// TIA Portal V20 export
// export: Created 2025-12-01T14:56:59.5537053Z, ExportSetting None, DisplayName Totally Integrated Automation Portal, DisplayVersion V20 Update 3, DisplayName TIA Portal Openness, DisplayVersion V20 Update 3, DisplayName TIA Portal Version Control Interface, DisplayVersion V20 Update 3, DisplayName STEP 7 Professional, DisplayVersion V20 Update 3, DisplayName STEP 7 Safety, DisplayVersion V20 Update 2, DisplayName WinCC Basic/Comfort/Advanced, DisplayVersion V20 Update 3, DisplayName WinCC Professional, DisplayVersion V20 Update 3, DisplayName WinCC Unified, DisplayVersion V20 Update 3
FUNCTION "FC421_TL_ZPA_Tarjeta_CB_E1E3S1S3" : Void   // FC421, LAD
{ S7_Optimized_Access := 'FALSE' }
AUTHOR : TLigero
NAME : 20160208
VERSION : 3.1
// FECHA:    27/07/2014  AUTOR: G.Martin
// INSTALACION: Magyar Posta
// //////////////////////////////////
// // Registro Incidencias   ////////
// //////////////////////////////////
// FECHA:21/10/14   AUTOR MODIFICACION: N.Rodriguez
// DESCRIPCION: 
// Adaptación de la función al estandar actual
// 
// FECHA:   AUTOR MODIFICACION: 
// DESCRIPCION:
// stored: AutoNumber false, SetENOAutomatically false
   VAR_INPUT
      Mesa : UInt;
      En_Tension : Bool;
      Phs_Tx_E1 : Bool;
      Phs_Tx_E3 : Bool;
      Avance_E1 : Bool;
      Avance_E3 : Bool;
      Termico_Tx : Bool;   // Señal de termico OK
      Simul_Mx : Bool;
      Invertir_Sentido : Bool;   // OFF sentido 1-3 a ON sentido 3-1
      AVTF_Ent_M1 : Bool;
      AVTF_Ent_M3 : Bool;
      PTF_Sal_M3 : Bool;
      NXT_Avance_M3 : Bool;
      PTF_Sal_M1 : Bool;
      NXT_Avance_M1 : Bool;
      V_CNT_pHsMx_E1 : UDInt;
      V_CNT_pHsMx_E3 : UDInt;
      V_Gap_E1 : UDInt;
      V_Gap_E3 : UDInt;
      V_Paro : UDInt;
      V_TOut_Tx_Mx : UDInt;
      V_Salida : UDInt;
   END_VAR
   VAR_OUTPUT
      PTF_Ent_M1 : Bool;
      PTF_Ent_M3 : Bool;
      AVTF_Sal_M1 : Bool;
      NXT_Descarga_Act_M1 : Bool;
      AVTF_Sal_M3 : Bool;
      NXT_Descarga_Act_M3 : Bool;
   END_VAR
   VAR_IN_OUT
      Mem_CNT_Salida : Bool;
      Mem_CNT_Tmp_Paro_Tx : Bool;
      MAUX_FP_Marcha : Bool;
      MAUX_FN_PHS : Bool;
      MAUX_FP_Direc : Bool;
      MAUX_FN_Direc : Bool;
   END_VAR
   VAR_TEMP
      OK_Avance : Bool;
      fp_Marcha : Bool;
      fn_phs_tx : Bool;
      fp_phs_tx : Bool;
      Mem_CNT_Centrado : Bool;
      Mem_CNT_Gap : Bool;
      fp_direc : Bool;
      fn_direc : Bool;
      Error_Atasco : Bool;
      Error_Atasco_Inv : Bool;
      TEMP_NXT_AVTF : Bool;
      TEMP_NXT_AVTF_Inv : Bool;
      ok_tension : Bool;
   END_VAR
   VAR_TEMP   // added for the SCL form of the ladder/FBD networks
      _w1 : Bool;
      _w2 : Bool;
   END_VAR
BEGIN

REGION Network 1: Marca General Error
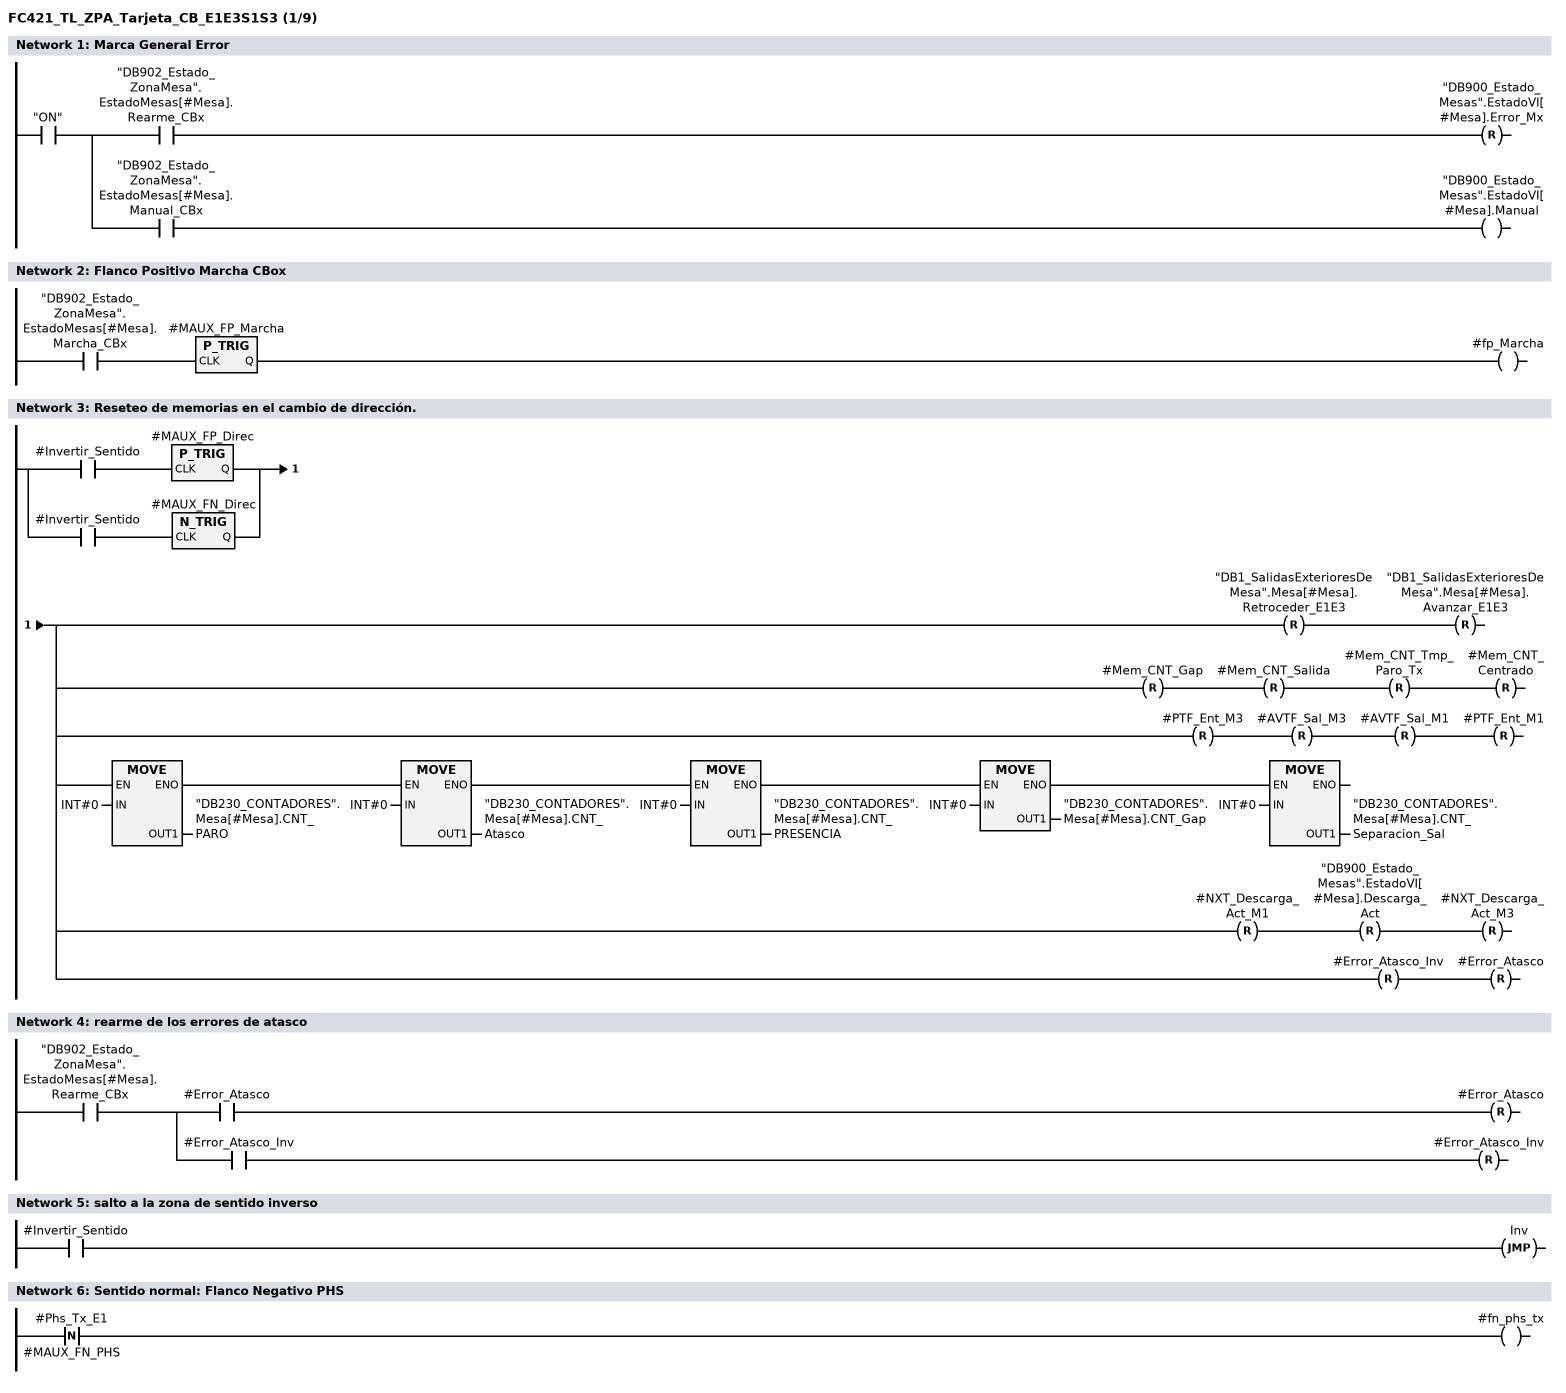
   RUNG wire#powerrail
      Contact( "ON" )
      wire#w1
      Contact( "DB902_Estado_ZonaMesa".EstadoMesas[#Mesa].Rearme_CBx )
      R_Coil( "DB900_Estado_Mesas".EstadoVI[#Mesa].Error_Mx )
   END_RUNG
   RUNG wire#w1
      Contact( "DB902_Estado_ZonaMesa".EstadoMesas[#Mesa].Manual_CBx )
      Coil( "DB900_Estado_Mesas".EstadoVI[#Mesa].Manual )
   END_RUNG
   // the same network as SCL:
   IF "ON" AND "DB902_Estado_ZonaMesa".EstadoMesas[#Mesa].Rearme_CBx THEN
       "DB900_Estado_Mesas".EstadoVI[#Mesa].Error_Mx := FALSE;
   END_IF;
   "DB900_Estado_Mesas".EstadoVI[#Mesa].Manual := "ON" AND "DB902_Estado_ZonaMesa".EstadoMesas[#Mesa].Manual_CBx;
END_REGION

REGION Network 2: Flanco Positivo Marcha CBox
   RUNG wire#powerrail
      Contact( "DB902_Estado_ZonaMesa".EstadoMesas[#Mesa].Marcha_CBx )
      P_Trig( #MAUX_FP_Marcha )
      Coil( #fp_Marcha )
   END_RUNG
   // the same network as SCL:
   #_w1 := "DB902_Estado_ZonaMesa".EstadoMesas[#Mesa].Marcha_CBx AND NOT #MAUX_FP_Marcha;   // rising edge
   #MAUX_FP_Marcha := "DB902_Estado_ZonaMesa".EstadoMesas[#Mesa].Marcha_CBx;
   #fp_Marcha := #_w1;
END_REGION

REGION Network 3: Reseteo de memorias en el cambio de dirección.
   RUNG wire#powerrail
      Contact( #Invertir_Sentido )
      P_Trig( #MAUX_FP_Direc )
      wire#w1
      R_Coil( "DB1_SalidasExterioresDeMesa".Mesa[#Mesa].Retroceder_E1E3 )
      R_Coil( "DB1_SalidasExterioresDeMesa".Mesa[#Mesa].Avanzar_E1E3 )
   END_RUNG
   RUNG wire#powerrail
      Contact( #Invertir_Sentido )
      N_Trig( #MAUX_FN_Direc )
   END_RUNG wire#w1
   RUNG wire#w1
      R_Coil( #Mem_CNT_Gap )
      R_Coil( #Mem_CNT_Salida )
      R_Coil( #Mem_CNT_Tmp_Paro_Tx )
      R_Coil( #Mem_CNT_Centrado )
   END_RUNG
   RUNG wire#w1
      R_Coil( #PTF_Ent_M3 )
      R_Coil( #AVTF_Sal_M3 )
      R_Coil( #AVTF_Sal_M1 )
      R_Coil( #PTF_Ent_M1 )
   END_RUNG
   RUNG wire#w1
      { S7_GenerateENO := "TRUE" } Move(in := INT#0, out1 => "DB230_CONTADORES".Mesa[#Mesa].CNT_PARO)
      { S7_GenerateENO := "TRUE" } Move(in := INT#0, out1 => "DB230_CONTADORES".Mesa[#Mesa].CNT_Atasco)
      { S7_GenerateENO := "TRUE" } Move(in := INT#0, out1 => "DB230_CONTADORES".Mesa[#Mesa].CNT_PRESENCIA)
      { S7_GenerateENO := "TRUE" } Move(in := INT#0, out1 => "DB230_CONTADORES".Mesa[#Mesa].CNT_Gap)
      { S7_GenerateENO := "TRUE" } Move(in := INT#0, out1 => "DB230_CONTADORES".Mesa[#Mesa].CNT_Separacion_Sal)
   END_RUNG
   RUNG wire#w1
      R_Coil( #NXT_Descarga_Act_M1 )
      R_Coil( "DB900_Estado_Mesas".EstadoVI[#Mesa].Descarga_Act )
      R_Coil( #NXT_Descarga_Act_M3 )
   END_RUNG
   RUNG wire#w1
      R_Coil( #Error_Atasco_Inv )
      R_Coil( #Error_Atasco )
   END_RUNG
   // the same network as SCL:
   // ENO of a box is taken as its EN; it also drops when the box reports an error
   #_w1 := #Invertir_Sentido AND NOT #MAUX_FP_Direc;   // rising edge
   #MAUX_FP_Direc := #Invertir_Sentido;
   #_w2 := NOT #Invertir_Sentido AND #MAUX_FN_Direc;   // falling edge
   #MAUX_FN_Direc := #Invertir_Sentido;
   IF #_w1 OR #_w2 THEN
       "DB1_SalidasExterioresDeMesa".Mesa[#Mesa].Retroceder_E1E3 := FALSE;
       "DB1_SalidasExterioresDeMesa".Mesa[#Mesa].Avanzar_E1E3 := FALSE;
       #Mem_CNT_Gap := FALSE;
       #Mem_CNT_Salida := FALSE;
       #Mem_CNT_Tmp_Paro_Tx := FALSE;
       #Mem_CNT_Centrado := FALSE;
       #PTF_Ent_M3 := FALSE;
       #AVTF_Sal_M3 := FALSE;
       #AVTF_Sal_M1 := FALSE;
       #PTF_Ent_M1 := FALSE;
       "DB230_CONTADORES".Mesa[#Mesa].CNT_PARO := INT#0;
       "DB230_CONTADORES".Mesa[#Mesa].CNT_Atasco := INT#0;
       "DB230_CONTADORES".Mesa[#Mesa].CNT_PRESENCIA := INT#0;
       "DB230_CONTADORES".Mesa[#Mesa].CNT_Gap := INT#0;
       "DB230_CONTADORES".Mesa[#Mesa].CNT_Separacion_Sal := INT#0;
       #NXT_Descarga_Act_M1 := FALSE;
       "DB900_Estado_Mesas".EstadoVI[#Mesa].Descarga_Act := FALSE;
       #NXT_Descarga_Act_M3 := FALSE;
       #Error_Atasco_Inv := FALSE;
       #Error_Atasco := FALSE;
   END_IF;
END_REGION

REGION Network 4: rearme de los errores de atasco
   RUNG wire#powerrail
      Contact( "DB902_Estado_ZonaMesa".EstadoMesas[#Mesa].Rearme_CBx )
      wire#w1
      Contact( #Error_Atasco )
      R_Coil( #Error_Atasco )
   END_RUNG
   RUNG wire#w1
      Contact( #Error_Atasco_Inv )
      R_Coil( #Error_Atasco_Inv )
   END_RUNG
   // the same network as SCL:
   IF "DB902_Estado_ZonaMesa".EstadoMesas[#Mesa].Rearme_CBx AND #Error_Atasco THEN
       #Error_Atasco := FALSE;
   END_IF;
   IF "DB902_Estado_ZonaMesa".EstadoMesas[#Mesa].Rearme_CBx AND #Error_Atasco_Inv THEN
       #Error_Atasco_Inv := FALSE;
   END_IF;
END_REGION

REGION Network 5: salto a la zona de sentido inverso
   RUNG wire#powerrail
      Contact( #Invertir_Sentido )
      JumpCoil( Inv )
   END_RUNG
   // the same network as SCL:
   IF #Invertir_Sentido THEN GOTO Inv; END_IF;
END_REGION

REGION Network 6: Sentido normal: Flanco Negativo PHS
   RUNG wire#powerrail
      N_Contact(operand := #Phs_Tx_E1, bit := #MAUX_FN_PHS)
      Coil( #fn_phs_tx )
   END_RUNG
   // the same network as SCL:
   #_w1 := NOT #Phs_Tx_E1 AND #MAUX_FN_PHS;   // falling edge of #Phs_Tx_E1
   #MAUX_FN_PHS := #Phs_Tx_E1;
   #fn_phs_tx := #_w1;
END_REGION

REGION Network 7: En Tension
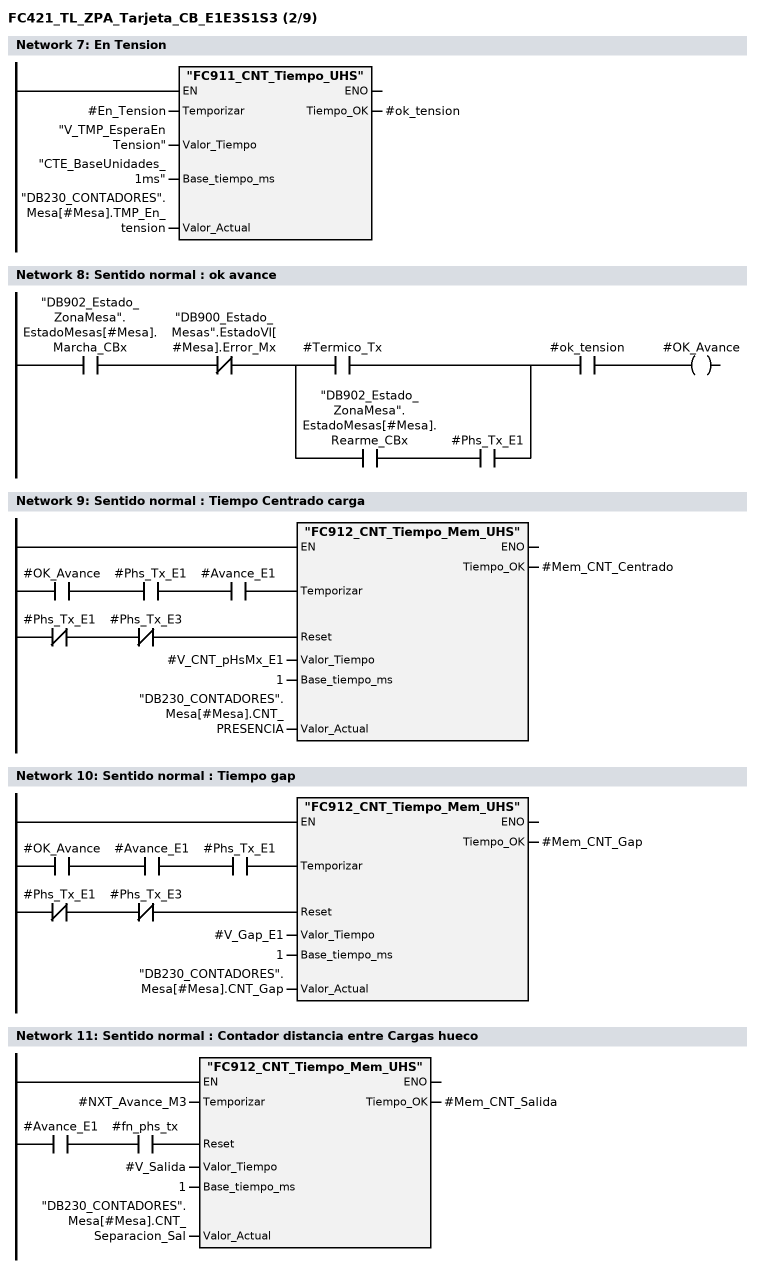
   RUNG wire#powerrail
      "FC911_CNT_Tiempo_UHS"(Temporizar := #En_Tension, Valor_Tiempo := "V_TMP_EsperaEnTension", Base_tiempo_ms := "CTE_BaseUnidades_1ms", Valor_Actual := "DB230_CONTADORES".Mesa[#Mesa].TMP_En_tension, Tiempo_OK => #ok_tension)
   END_RUNG
   // the same network as SCL:
   "FC911_CNT_Tiempo_UHS"(Temporizar := #En_Tension,
                          Valor_Tiempo := "V_TMP_EsperaEnTension",
                          Base_tiempo_ms := "CTE_BaseUnidades_1ms",
                          Valor_Actual := "DB230_CONTADORES".Mesa[#Mesa].TMP_En_tension,
                          Tiempo_OK => #ok_tension);
END_REGION

REGION Network 8: Sentido normal : ok avance
   RUNG wire#powerrail
      Contact( "DB902_Estado_ZonaMesa".EstadoMesas[#Mesa].Marcha_CBx )
      I_Contact( "DB900_Estado_Mesas".EstadoVI[#Mesa].Error_Mx )
      wire#w1
      Contact( #Termico_Tx )
      wire#w2
      Contact( #ok_tension )
      Coil( #OK_Avance )
   END_RUNG
   RUNG wire#w1
      Contact( "DB902_Estado_ZonaMesa".EstadoMesas[#Mesa].Rearme_CBx )
      Contact( #Phs_Tx_E1 )
   END_RUNG wire#w2
   // the same network as SCL:
   #OK_Avance := "DB902_Estado_ZonaMesa".EstadoMesas[#Mesa].Marcha_CBx AND NOT "DB900_Estado_Mesas".EstadoVI[#Mesa].Error_Mx AND (#Termico_Tx OR ("DB902_Estado_ZonaMesa".EstadoMesas[#Mesa].Rearme_CBx AND #Phs_Tx_E1)) AND #ok_tension;
END_REGION

REGION Network 9: Sentido normal : Tiempo Centrado carga
   RUNG wire#powerrail
      "FC912_CNT_Tiempo_Mem_UHS"(Temporizar := wire#w1, Reset := wire#w2, Valor_Tiempo := #V_CNT_pHsMx_E1, Base_tiempo_ms := 1, Valor_Actual := "DB230_CONTADORES".Mesa[#Mesa].CNT_PRESENCIA, Tiempo_OK => #Mem_CNT_Centrado)
   END_RUNG
   RUNG wire#powerrail
      Contact( #OK_Avance )
      Contact( #Phs_Tx_E1 )
      Contact( #Avance_E1 )
   END_RUNG wire#w1
   RUNG wire#powerrail
      I_Contact( #Phs_Tx_E1 )
      I_Contact( #Phs_Tx_E3 )
   END_RUNG wire#w2
   // the same network as SCL:
   "FC912_CNT_Tiempo_Mem_UHS"(Temporizar := #OK_Avance AND #Phs_Tx_E1 AND #Avance_E1,
                           Reset := NOT #Phs_Tx_E1 AND NOT #Phs_Tx_E3,
                           Valor_Tiempo := #V_CNT_pHsMx_E1,
                           Base_tiempo_ms := 1,
                           Valor_Actual := "DB230_CONTADORES".Mesa[#Mesa].CNT_PRESENCIA,
                           Tiempo_OK => #Mem_CNT_Centrado);
END_REGION

REGION Network 10: Sentido normal : Tiempo gap
   RUNG wire#powerrail
      "FC912_CNT_Tiempo_Mem_UHS"(Temporizar := wire#w1, Reset := wire#w2, Valor_Tiempo := #V_Gap_E1, Base_tiempo_ms := 1, Valor_Actual := "DB230_CONTADORES".Mesa[#Mesa].CNT_Gap, Tiempo_OK => #Mem_CNT_Gap)
   END_RUNG
   RUNG wire#powerrail
      Contact( #OK_Avance )
      Contact( #Avance_E1 )
      Contact( #Phs_Tx_E1 )
   END_RUNG wire#w1
   RUNG wire#powerrail
      I_Contact( #Phs_Tx_E1 )
      I_Contact( #Phs_Tx_E3 )
   END_RUNG wire#w2
   // the same network as SCL:
   "FC912_CNT_Tiempo_Mem_UHS"(Temporizar := #OK_Avance AND #Avance_E1 AND #Phs_Tx_E1,
                           Reset := NOT #Phs_Tx_E1 AND NOT #Phs_Tx_E3,
                           Valor_Tiempo := #V_Gap_E1,
                           Base_tiempo_ms := 1,
                           Valor_Actual := "DB230_CONTADORES".Mesa[#Mesa].CNT_Gap,
                           Tiempo_OK => #Mem_CNT_Gap);
END_REGION

REGION Network 11: Sentido normal : Contador distancia entre Cargas hueco
   RUNG wire#powerrail
      "FC912_CNT_Tiempo_Mem_UHS"(Reset := wire#w1, Temporizar := #NXT_Avance_M3, Valor_Tiempo := #V_Salida, Base_tiempo_ms := 1, Valor_Actual := "DB230_CONTADORES".Mesa[#Mesa].CNT_Separacion_Sal, Tiempo_OK => #Mem_CNT_Salida)
   END_RUNG
   RUNG wire#powerrail
      Contact( #Avance_E1 )
      Contact( #fn_phs_tx )
   END_RUNG wire#w1
   // the same network as SCL:
   "FC912_CNT_Tiempo_Mem_UHS"(Temporizar := #NXT_Avance_M3,
                           Reset := #Avance_E1 AND #fn_phs_tx,
                           Valor_Tiempo := #V_Salida,
                           Base_tiempo_ms := 1,
                           Valor_Actual := "DB230_CONTADORES".Mesa[#Mesa].CNT_Separacion_Sal,
                           Tiempo_OK => #Mem_CNT_Salida);
END_REGION

REGION Network 12: Sentido normal : temporizador de paro
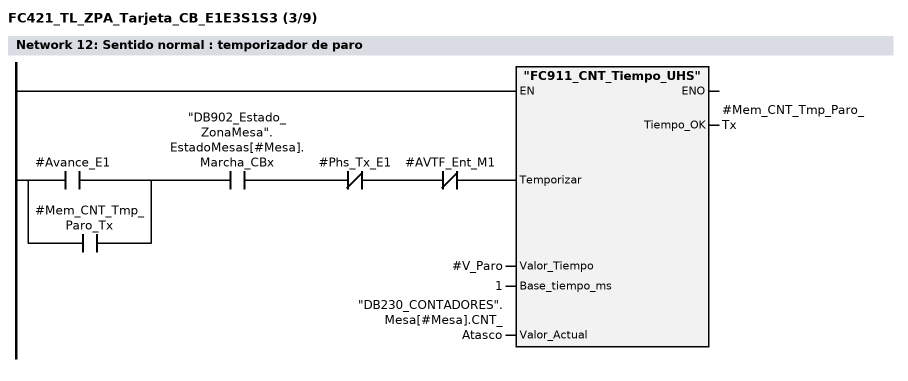
   RUNG wire#powerrail
      "FC911_CNT_Tiempo_UHS"(Temporizar := wire#w2, Valor_Tiempo := #V_Paro, Base_tiempo_ms := 1, Valor_Actual := "DB230_CONTADORES".Mesa[#Mesa].CNT_Atasco, Tiempo_OK => #Mem_CNT_Tmp_Paro_Tx)
   END_RUNG
   RUNG wire#powerrail
      Contact( #Avance_E1 )
      wire#w1
      Contact( "DB902_Estado_ZonaMesa".EstadoMesas[#Mesa].Marcha_CBx )
      I_Contact( #Phs_Tx_E1 )
      I_Contact( #AVTF_Ent_M1 )
   END_RUNG wire#w2
   RUNG wire#powerrail
      Contact( #Mem_CNT_Tmp_Paro_Tx )
   END_RUNG wire#w1
   // the same network as SCL:
   "FC911_CNT_Tiempo_UHS"(Temporizar := (#Avance_E1 OR #Mem_CNT_Tmp_Paro_Tx) AND "DB902_Estado_ZonaMesa".EstadoMesas[#Mesa].Marcha_CBx AND NOT #Phs_Tx_E1 AND NOT #AVTF_Ent_M1,
                          Valor_Tiempo := #V_Paro,
                          Base_tiempo_ms := 1,
                          Valor_Actual := "DB230_CONTADORES".Mesa[#Mesa].CNT_Atasco,
                          Tiempo_OK => #Mem_CNT_Tmp_Paro_Tx);
END_REGION

REGION Network 13: Sentido normal : avance 13
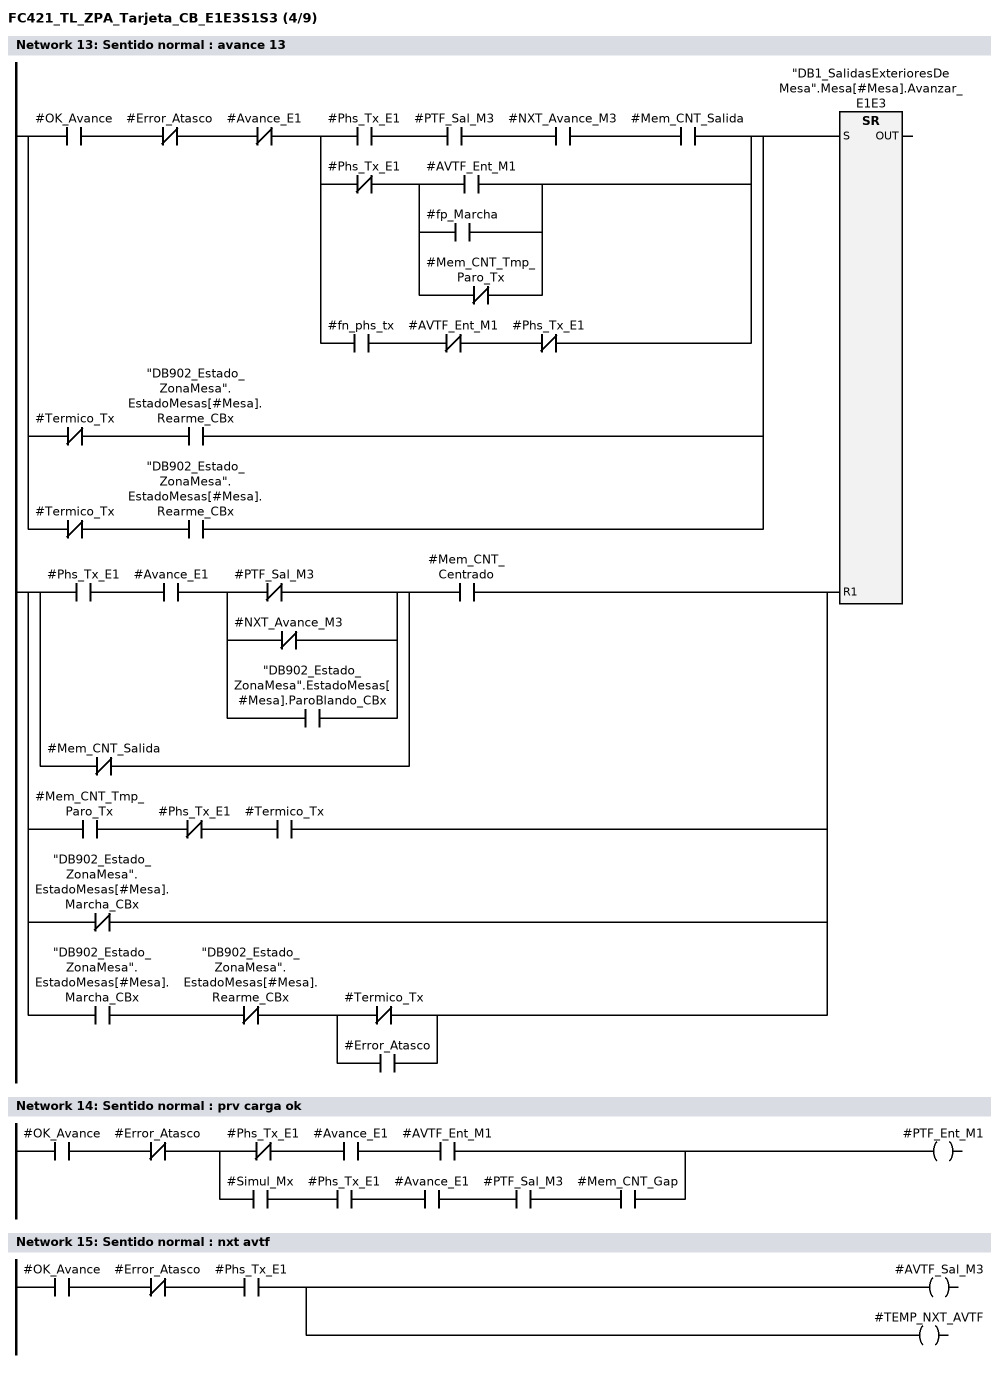
   RUNG wire#powerrail
      Contact( #OK_Avance )
      I_Contact( #Error_Atasco )
      I_Contact( #Avance_E1 )
      wire#w1
      Contact( #Phs_Tx_E1 )
      Contact( #PTF_Sal_M3 )
      Contact( #NXT_Avance_M3 )
      Contact( #Mem_CNT_Salida )
      wire#w2
      S_SR(operand := "DB1_SalidasExterioresDeMesa".Mesa[#Mesa].Avanzar_E1E3, r1 := wire#w7)
   END_RUNG
   RUNG wire#w1
      I_Contact( #Phs_Tx_E1 )
      wire#w3
      Contact( #AVTF_Ent_M1 )
   END_RUNG wire#w2
   RUNG wire#w3
      Contact( #fp_Marcha )
   END_RUNG wire#w2
   RUNG wire#w3
      I_Contact( #Mem_CNT_Tmp_Paro_Tx )
   END_RUNG wire#w2
   RUNG wire#w1
      Contact( #fn_phs_tx )
      I_Contact( #AVTF_Ent_M1 )
      I_Contact( #Phs_Tx_E1 )
   END_RUNG wire#w2
   RUNG wire#powerrail
      I_Contact( #Termico_Tx )
      Contact( "DB902_Estado_ZonaMesa".EstadoMesas[#Mesa].Rearme_CBx )
   END_RUNG wire#w2
   RUNG wire#powerrail
      I_Contact( #Termico_Tx )
      Contact( "DB902_Estado_ZonaMesa".EstadoMesas[#Mesa].Rearme_CBx )
   END_RUNG wire#w2
   RUNG wire#powerrail
      Contact( #Phs_Tx_E1 )
      Contact( #Avance_E1 )
      wire#w4
      I_Contact( #PTF_Sal_M3 )
      wire#w5
      Contact( #Mem_CNT_Centrado )
   END_RUNG wire#w7
   RUNG wire#w4
      I_Contact( #NXT_Avance_M3 )
   END_RUNG wire#w5
   RUNG wire#w4
      Contact( "DB902_Estado_ZonaMesa".EstadoMesas[#Mesa].ParoBlando_CBx )
   END_RUNG wire#w5
   RUNG wire#powerrail
      I_Contact( #Mem_CNT_Salida )
   END_RUNG wire#w5
   RUNG wire#powerrail
      Contact( #Mem_CNT_Tmp_Paro_Tx )
      I_Contact( #Phs_Tx_E1 )
      Contact( #Termico_Tx )
   END_RUNG wire#w7
   RUNG wire#powerrail
      I_Contact( "DB902_Estado_ZonaMesa".EstadoMesas[#Mesa].Marcha_CBx )
   END_RUNG wire#w7
   RUNG wire#powerrail
      Contact( "DB902_Estado_ZonaMesa".EstadoMesas[#Mesa].Marcha_CBx )
      I_Contact( "DB902_Estado_ZonaMesa".EstadoMesas[#Mesa].Rearme_CBx )
      wire#w6
      I_Contact( #Termico_Tx )
   END_RUNG wire#w7
   RUNG wire#w6
      Contact( #Error_Atasco )
   END_RUNG wire#w7
   // the same network as SCL:
   #_w1 := (((#Phs_Tx_E1 AND #Avance_E1 AND (NOT #PTF_Sal_M3 OR NOT #NXT_Avance_M3 OR "DB902_Estado_ZonaMesa".EstadoMesas[#Mesa].ParoBlando_CBx)) OR NOT #Mem_CNT_Salida) AND #Mem_CNT_Centrado) OR (#Mem_CNT_Tmp_Paro_Tx AND NOT #Phs_Tx_E1 AND #Termico_Tx) OR NOT "DB902_Estado_ZonaMesa".EstadoMesas[#Mesa].Marcha_CBx OR ("DB902_Estado_ZonaMesa".EstadoMesas[#Mesa].Marcha_CBx AND NOT "DB902_Estado_ZonaMesa".EstadoMesas[#Mesa].Rearme_CBx AND (NOT #Termico_Tx OR #Error_Atasco));
   IF (#OK_Avance AND NOT #Error_Atasco AND NOT #Avance_E1 AND ((#Phs_Tx_E1 AND #PTF_Sal_M3 AND #NXT_Avance_M3 AND #Mem_CNT_Salida) OR (NOT #Phs_Tx_E1 AND (#AVTF_Ent_M1 OR #fp_Marcha OR NOT #Mem_CNT_Tmp_Paro_Tx)) OR (#fn_phs_tx AND NOT #AVTF_Ent_M1 AND NOT #Phs_Tx_E1))) OR (NOT #Termico_Tx AND "DB902_Estado_ZonaMesa".EstadoMesas[#Mesa].Rearme_CBx) OR (NOT #Termico_Tx AND "DB902_Estado_ZonaMesa".EstadoMesas[#Mesa].Rearme_CBx) THEN
       "DB1_SalidasExterioresDeMesa".Mesa[#Mesa].Avanzar_E1E3 := TRUE;   // SR flip-flop
   END_IF;
   IF #_w1 THEN "DB1_SalidasExterioresDeMesa".Mesa[#Mesa].Avanzar_E1E3 := FALSE; END_IF;
END_REGION

REGION Network 14: Sentido normal : prv carga ok
   RUNG wire#powerrail
      Contact( #OK_Avance )
      I_Contact( #Error_Atasco )
      wire#w1
      I_Contact( #Phs_Tx_E1 )
      Contact( #Avance_E1 )
      Contact( #AVTF_Ent_M1 )
      wire#w2
      Coil( #PTF_Ent_M1 )
   END_RUNG
   RUNG wire#w1
      Contact( #Simul_Mx )
      Contact( #Phs_Tx_E1 )
      Contact( #Avance_E1 )
      Contact( #PTF_Sal_M3 )
      Contact( #Mem_CNT_Gap )
   END_RUNG wire#w2
   // the same network as SCL:
   #PTF_Ent_M1 := #OK_Avance AND NOT #Error_Atasco AND ((NOT #Phs_Tx_E1 AND #Avance_E1 AND #AVTF_Ent_M1) OR (#Simul_Mx AND #Phs_Tx_E1 AND #Avance_E1 AND #PTF_Sal_M3 AND #Mem_CNT_Gap));
END_REGION

REGION Network 15: Sentido normal : nxt avtf
   RUNG wire#powerrail
      Contact( #OK_Avance )
      I_Contact( #Error_Atasco )
      Contact( #Phs_Tx_E1 )
      wire#w1
      Coil( #AVTF_Sal_M3 )
   END_RUNG
   RUNG wire#w1
      Coil( #TEMP_NXT_AVTF )
   END_RUNG
   // the same network as SCL:
   #AVTF_Sal_M3 := #OK_Avance AND NOT #Error_Atasco AND #Phs_Tx_E1;
   #TEMP_NXT_AVTF := #AVTF_Sal_M3;
END_REGION

REGION Network 16: Sentido normal : nxt descarga activa
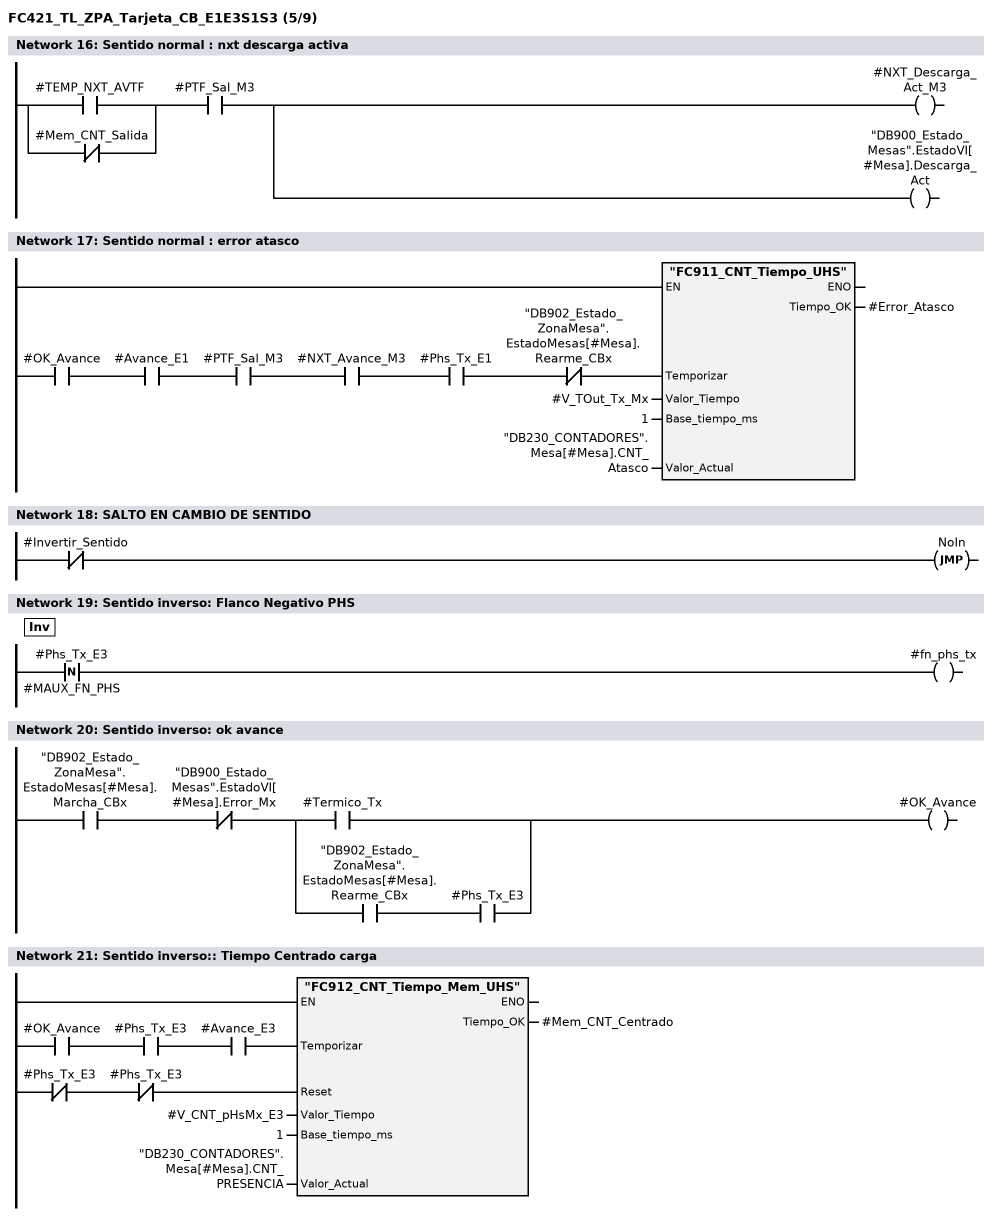
   RUNG wire#powerrail
      Contact( #TEMP_NXT_AVTF )
      wire#w1
      Contact( #PTF_Sal_M3 )
      wire#w2
      Coil( #NXT_Descarga_Act_M3 )
   END_RUNG
   RUNG wire#powerrail
      I_Contact( #Mem_CNT_Salida )
   END_RUNG wire#w1
   RUNG wire#w2
      Coil( "DB900_Estado_Mesas".EstadoVI[#Mesa].Descarga_Act )
   END_RUNG
   // the same network as SCL:
   #NXT_Descarga_Act_M3 := (#TEMP_NXT_AVTF OR NOT #Mem_CNT_Salida) AND #PTF_Sal_M3;
   "DB900_Estado_Mesas".EstadoVI[#Mesa].Descarga_Act := #NXT_Descarga_Act_M3;
END_REGION

REGION Network 17: Sentido normal : error atasco
   RUNG wire#powerrail
      "FC911_CNT_Tiempo_UHS"(Temporizar := wire#w1, Valor_Tiempo := #V_TOut_Tx_Mx, Base_tiempo_ms := 1, Valor_Actual := "DB230_CONTADORES".Mesa[#Mesa].CNT_Atasco, Tiempo_OK => #Error_Atasco)
   END_RUNG
   RUNG wire#powerrail
      Contact( #OK_Avance )
      Contact( #Avance_E1 )
      Contact( #PTF_Sal_M3 )
      Contact( #NXT_Avance_M3 )
      Contact( #Phs_Tx_E1 )
      I_Contact( "DB902_Estado_ZonaMesa".EstadoMesas[#Mesa].Rearme_CBx )
   END_RUNG wire#w1
   // the same network as SCL:
   "FC911_CNT_Tiempo_UHS"(Temporizar := #OK_Avance AND #Avance_E1 AND #PTF_Sal_M3 AND #NXT_Avance_M3 AND #Phs_Tx_E1 AND NOT "DB902_Estado_ZonaMesa".EstadoMesas[#Mesa].Rearme_CBx,
                          Valor_Tiempo := #V_TOut_Tx_Mx,
                          Base_tiempo_ms := 1,
                          Valor_Actual := "DB230_CONTADORES".Mesa[#Mesa].CNT_Atasco,
                          Tiempo_OK => #Error_Atasco);
END_REGION

REGION Network 18: SALTO EN CAMBIO DE SENTIDO
   RUNG wire#powerrail
      I_Contact( #Invertir_Sentido )
      JumpCoil( NoIn )
   END_RUNG
   // the same network as SCL:
   IF NOT #Invertir_Sentido THEN GOTO NoIn; END_IF;
END_REGION

REGION Network 19: Sentido inverso: Flanco Negativo PHS
   Label( Inv )
   RUNG wire#powerrail
      N_Contact(operand := #Phs_Tx_E3, bit := #MAUX_FN_PHS)
      Coil( #fn_phs_tx )
   END_RUNG
   // the same network as SCL:
   Inv:
   #_w1 := NOT #Phs_Tx_E3 AND #MAUX_FN_PHS;   // falling edge of #Phs_Tx_E3
   #MAUX_FN_PHS := #Phs_Tx_E3;
   #fn_phs_tx := #_w1;
END_REGION

REGION Network 20: Sentido inverso: ok avance
   RUNG wire#powerrail
      Contact( "DB902_Estado_ZonaMesa".EstadoMesas[#Mesa].Marcha_CBx )
      I_Contact( "DB900_Estado_Mesas".EstadoVI[#Mesa].Error_Mx )
      wire#w1
      Contact( #Termico_Tx )
      wire#w2
      Coil( #OK_Avance )
   END_RUNG
   RUNG wire#w1
      Contact( "DB902_Estado_ZonaMesa".EstadoMesas[#Mesa].Rearme_CBx )
      Contact( #Phs_Tx_E3 )
   END_RUNG wire#w2
   // the same network as SCL:
   #OK_Avance := "DB902_Estado_ZonaMesa".EstadoMesas[#Mesa].Marcha_CBx AND NOT "DB900_Estado_Mesas".EstadoVI[#Mesa].Error_Mx AND (#Termico_Tx OR ("DB902_Estado_ZonaMesa".EstadoMesas[#Mesa].Rearme_CBx AND #Phs_Tx_E3));
END_REGION

REGION Network 21: Sentido inverso:: Tiempo Centrado carga
   RUNG wire#powerrail
      "FC912_CNT_Tiempo_Mem_UHS"(Temporizar := wire#w1, Reset := wire#w2, Valor_Tiempo := #V_CNT_pHsMx_E3, Base_tiempo_ms := 1, Valor_Actual := "DB230_CONTADORES".Mesa[#Mesa].CNT_PRESENCIA, Tiempo_OK => #Mem_CNT_Centrado)
   END_RUNG
   RUNG wire#powerrail
      Contact( #OK_Avance )
      Contact( #Phs_Tx_E3 )
      Contact( #Avance_E3 )
   END_RUNG wire#w1
   RUNG wire#powerrail
      I_Contact( #Phs_Tx_E3 )
      I_Contact( #Phs_Tx_E3 )
   END_RUNG wire#w2
   // the same network as SCL:
   "FC912_CNT_Tiempo_Mem_UHS"(Temporizar := #OK_Avance AND #Phs_Tx_E3 AND #Avance_E3,
                           Reset := NOT #Phs_Tx_E3 AND NOT #Phs_Tx_E3,
                           Valor_Tiempo := #V_CNT_pHsMx_E3,
                           Base_tiempo_ms := 1,
                           Valor_Actual := "DB230_CONTADORES".Mesa[#Mesa].CNT_PRESENCIA,
                           Tiempo_OK => #Mem_CNT_Centrado);
END_REGION

REGION Network 22: Sentido inverso: Tiempo gap
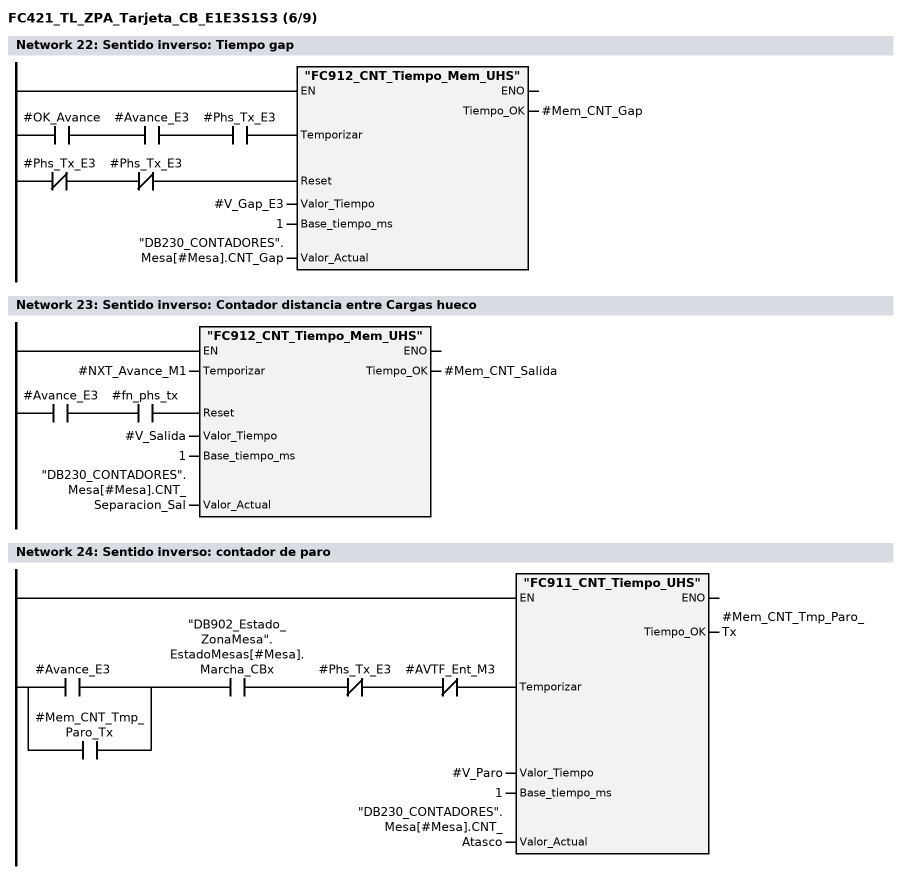
   RUNG wire#powerrail
      "FC912_CNT_Tiempo_Mem_UHS"(Temporizar := wire#w1, Reset := wire#w2, Valor_Tiempo := #V_Gap_E3, Base_tiempo_ms := 1, Valor_Actual := "DB230_CONTADORES".Mesa[#Mesa].CNT_Gap, Tiempo_OK => #Mem_CNT_Gap)
   END_RUNG
   RUNG wire#powerrail
      Contact( #OK_Avance )
      Contact( #Avance_E3 )
      Contact( #Phs_Tx_E3 )
   END_RUNG wire#w1
   RUNG wire#powerrail
      I_Contact( #Phs_Tx_E3 )
      I_Contact( #Phs_Tx_E3 )
   END_RUNG wire#w2
   // the same network as SCL:
   "FC912_CNT_Tiempo_Mem_UHS"(Temporizar := #OK_Avance AND #Avance_E3 AND #Phs_Tx_E3,
                           Reset := NOT #Phs_Tx_E3 AND NOT #Phs_Tx_E3,
                           Valor_Tiempo := #V_Gap_E3,
                           Base_tiempo_ms := 1,
                           Valor_Actual := "DB230_CONTADORES".Mesa[#Mesa].CNT_Gap,
                           Tiempo_OK => #Mem_CNT_Gap);
END_REGION

REGION Network 23: Sentido inverso: Contador distancia entre Cargas hueco
   RUNG wire#powerrail
      "FC912_CNT_Tiempo_Mem_UHS"(Reset := wire#w1, Temporizar := #NXT_Avance_M1, Valor_Tiempo := #V_Salida, Base_tiempo_ms := 1, Valor_Actual := "DB230_CONTADORES".Mesa[#Mesa].CNT_Separacion_Sal, Tiempo_OK => #Mem_CNT_Salida)
   END_RUNG
   RUNG wire#powerrail
      Contact( #Avance_E3 )
      Contact( #fn_phs_tx )
   END_RUNG wire#w1
   // the same network as SCL:
   "FC912_CNT_Tiempo_Mem_UHS"(Temporizar := #NXT_Avance_M1,
                           Reset := #Avance_E3 AND #fn_phs_tx,
                           Valor_Tiempo := #V_Salida,
                           Base_tiempo_ms := 1,
                           Valor_Actual := "DB230_CONTADORES".Mesa[#Mesa].CNT_Separacion_Sal,
                           Tiempo_OK => #Mem_CNT_Salida);
END_REGION

REGION Network 24: Sentido inverso: contador de paro
   RUNG wire#powerrail
      "FC911_CNT_Tiempo_UHS"(Temporizar := wire#w2, Valor_Tiempo := #V_Paro, Base_tiempo_ms := 1, Valor_Actual := "DB230_CONTADORES".Mesa[#Mesa].CNT_Atasco, Tiempo_OK => #Mem_CNT_Tmp_Paro_Tx)
   END_RUNG
   RUNG wire#powerrail
      Contact( #Avance_E3 )
      wire#w1
      Contact( "DB902_Estado_ZonaMesa".EstadoMesas[#Mesa].Marcha_CBx )
      I_Contact( #Phs_Tx_E3 )
      I_Contact( #AVTF_Ent_M3 )
   END_RUNG wire#w2
   RUNG wire#powerrail
      Contact( #Mem_CNT_Tmp_Paro_Tx )
   END_RUNG wire#w1
   // the same network as SCL:
   "FC911_CNT_Tiempo_UHS"(Temporizar := (#Avance_E3 OR #Mem_CNT_Tmp_Paro_Tx) AND "DB902_Estado_ZonaMesa".EstadoMesas[#Mesa].Marcha_CBx AND NOT #Phs_Tx_E3 AND NOT #AVTF_Ent_M3,
                          Valor_Tiempo := #V_Paro,
                          Base_tiempo_ms := 1,
                          Valor_Actual := "DB230_CONTADORES".Mesa[#Mesa].CNT_Atasco,
                          Tiempo_OK => #Mem_CNT_Tmp_Paro_Tx);
END_REGION

REGION Network 25: Sentido inverso: retroceso 1-3
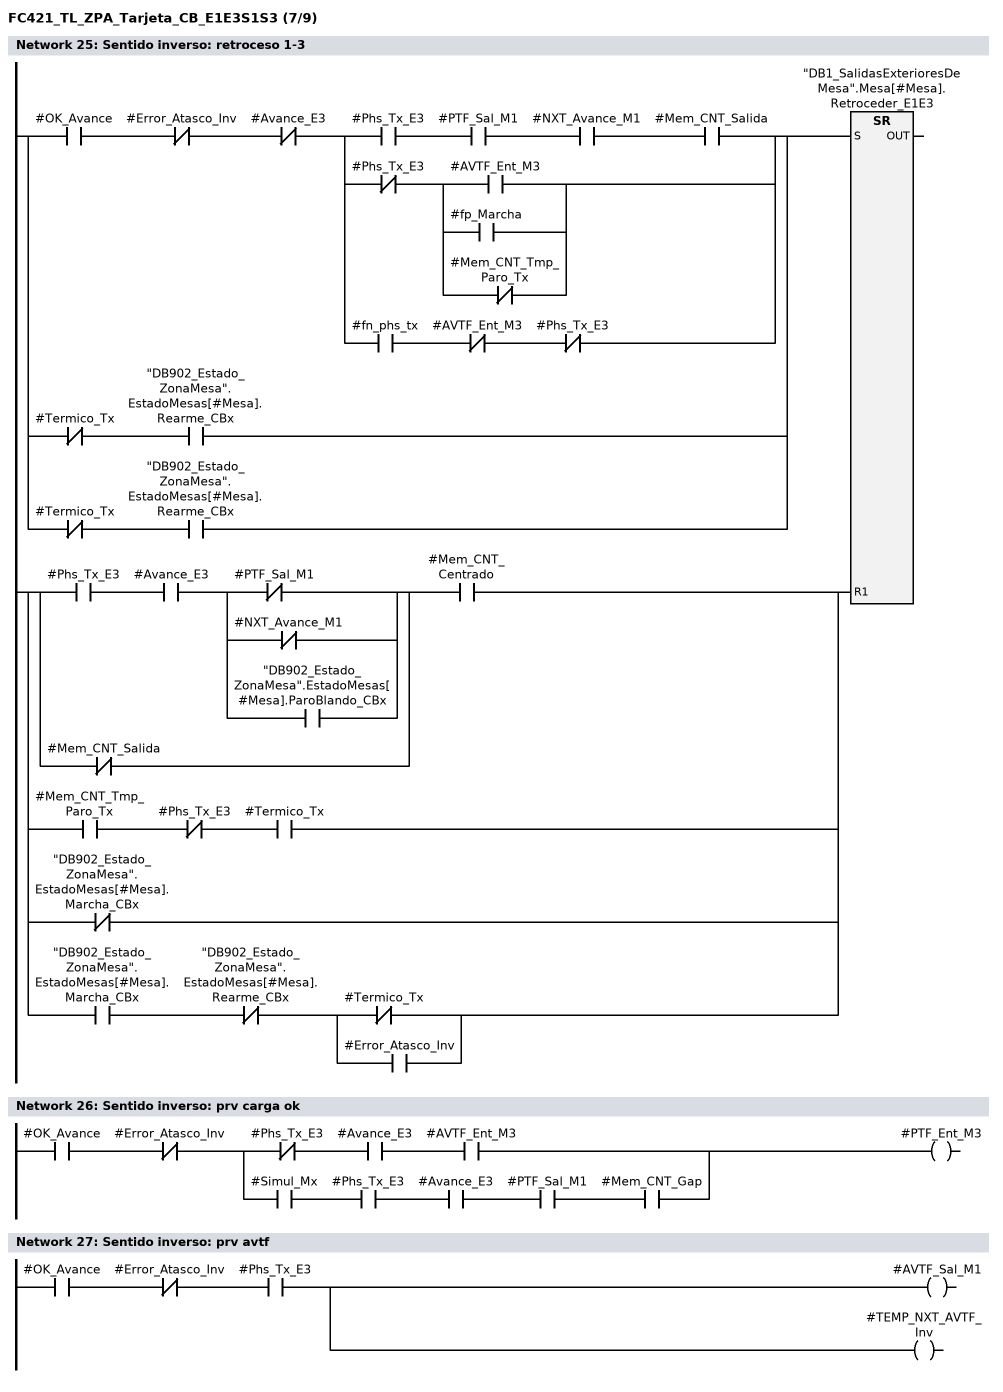
   RUNG wire#powerrail
      Contact( #OK_Avance )
      I_Contact( #Error_Atasco_Inv )
      I_Contact( #Avance_E3 )
      wire#w1
      Contact( #Phs_Tx_E3 )
      Contact( #PTF_Sal_M1 )
      Contact( #NXT_Avance_M1 )
      Contact( #Mem_CNT_Salida )
      wire#w2
      S_SR(operand := "DB1_SalidasExterioresDeMesa".Mesa[#Mesa].Retroceder_E1E3, r1 := wire#w7)
   END_RUNG
   RUNG wire#w1
      I_Contact( #Phs_Tx_E3 )
      wire#w3
      Contact( #AVTF_Ent_M3 )
   END_RUNG wire#w2
   RUNG wire#w3
      Contact( #fp_Marcha )
   END_RUNG wire#w2
   RUNG wire#w3
      I_Contact( #Mem_CNT_Tmp_Paro_Tx )
   END_RUNG wire#w2
   RUNG wire#w1
      Contact( #fn_phs_tx )
      I_Contact( #AVTF_Ent_M3 )
      I_Contact( #Phs_Tx_E3 )
   END_RUNG wire#w2
   RUNG wire#powerrail
      I_Contact( #Termico_Tx )
      Contact( "DB902_Estado_ZonaMesa".EstadoMesas[#Mesa].Rearme_CBx )
   END_RUNG wire#w2
   RUNG wire#powerrail
      I_Contact( #Termico_Tx )
      Contact( "DB902_Estado_ZonaMesa".EstadoMesas[#Mesa].Rearme_CBx )
   END_RUNG wire#w2
   RUNG wire#powerrail
      Contact( #Phs_Tx_E3 )
      Contact( #Avance_E3 )
      wire#w4
      I_Contact( #PTF_Sal_M1 )
      wire#w5
      Contact( #Mem_CNT_Centrado )
   END_RUNG wire#w7
   RUNG wire#w4
      I_Contact( #NXT_Avance_M1 )
   END_RUNG wire#w5
   RUNG wire#w4
      Contact( "DB902_Estado_ZonaMesa".EstadoMesas[#Mesa].ParoBlando_CBx )
   END_RUNG wire#w5
   RUNG wire#powerrail
      I_Contact( #Mem_CNT_Salida )
   END_RUNG wire#w5
   RUNG wire#powerrail
      Contact( #Mem_CNT_Tmp_Paro_Tx )
      I_Contact( #Phs_Tx_E3 )
      Contact( #Termico_Tx )
   END_RUNG wire#w7
   RUNG wire#powerrail
      I_Contact( "DB902_Estado_ZonaMesa".EstadoMesas[#Mesa].Marcha_CBx )
   END_RUNG wire#w7
   RUNG wire#powerrail
      Contact( "DB902_Estado_ZonaMesa".EstadoMesas[#Mesa].Marcha_CBx )
      I_Contact( "DB902_Estado_ZonaMesa".EstadoMesas[#Mesa].Rearme_CBx )
      wire#w6
      I_Contact( #Termico_Tx )
   END_RUNG wire#w7
   RUNG wire#w6
      Contact( #Error_Atasco_Inv )
   END_RUNG wire#w7
   // the same network as SCL:
   #_w1 := (((#Phs_Tx_E3 AND #Avance_E3 AND (NOT #PTF_Sal_M1 OR NOT #NXT_Avance_M1 OR "DB902_Estado_ZonaMesa".EstadoMesas[#Mesa].ParoBlando_CBx)) OR NOT #Mem_CNT_Salida) AND #Mem_CNT_Centrado) OR (#Mem_CNT_Tmp_Paro_Tx AND NOT #Phs_Tx_E3 AND #Termico_Tx) OR NOT "DB902_Estado_ZonaMesa".EstadoMesas[#Mesa].Marcha_CBx OR ("DB902_Estado_ZonaMesa".EstadoMesas[#Mesa].Marcha_CBx AND NOT "DB902_Estado_ZonaMesa".EstadoMesas[#Mesa].Rearme_CBx AND (NOT #Termico_Tx OR #Error_Atasco_Inv));
   IF (#OK_Avance AND NOT #Error_Atasco_Inv AND NOT #Avance_E3 AND ((#Phs_Tx_E3 AND #PTF_Sal_M1 AND #NXT_Avance_M1 AND #Mem_CNT_Salida) OR (NOT #Phs_Tx_E3 AND (#AVTF_Ent_M3 OR #fp_Marcha OR NOT #Mem_CNT_Tmp_Paro_Tx)) OR (#fn_phs_tx AND NOT #AVTF_Ent_M3 AND NOT #Phs_Tx_E3))) OR (NOT #Termico_Tx AND "DB902_Estado_ZonaMesa".EstadoMesas[#Mesa].Rearme_CBx) OR (NOT #Termico_Tx AND "DB902_Estado_ZonaMesa".EstadoMesas[#Mesa].Rearme_CBx) THEN
       "DB1_SalidasExterioresDeMesa".Mesa[#Mesa].Retroceder_E1E3 := TRUE;   // SR flip-flop
   END_IF;
   IF #_w1 THEN "DB1_SalidasExterioresDeMesa".Mesa[#Mesa].Retroceder_E1E3 := FALSE; END_IF;
END_REGION

REGION Network 26: Sentido inverso: prv carga ok
   RUNG wire#powerrail
      Contact( #OK_Avance )
      I_Contact( #Error_Atasco_Inv )
      wire#w1
      I_Contact( #Phs_Tx_E3 )
      Contact( #Avance_E3 )
      Contact( #AVTF_Ent_M3 )
      wire#w2
      Coil( #PTF_Ent_M3 )
   END_RUNG
   RUNG wire#w1
      Contact( #Simul_Mx )
      Contact( #Phs_Tx_E3 )
      Contact( #Avance_E3 )
      Contact( #PTF_Sal_M1 )
      Contact( #Mem_CNT_Gap )
   END_RUNG wire#w2
   // the same network as SCL:
   #PTF_Ent_M3 := #OK_Avance AND NOT #Error_Atasco_Inv AND ((NOT #Phs_Tx_E3 AND #Avance_E3 AND #AVTF_Ent_M3) OR (#Simul_Mx AND #Phs_Tx_E3 AND #Avance_E3 AND #PTF_Sal_M1 AND #Mem_CNT_Gap));
END_REGION

REGION Network 27: Sentido inverso: prv avtf
   RUNG wire#powerrail
      Contact( #OK_Avance )
      I_Contact( #Error_Atasco_Inv )
      Contact( #Phs_Tx_E3 )
      wire#w1
      Coil( #AVTF_Sal_M1 )
   END_RUNG
   RUNG wire#w1
      Coil( #TEMP_NXT_AVTF_Inv )
   END_RUNG
   // the same network as SCL:
   #AVTF_Sal_M1 := #OK_Avance AND NOT #Error_Atasco_Inv AND #Phs_Tx_E3;
   #TEMP_NXT_AVTF_Inv := #AVTF_Sal_M1;
END_REGION

REGION Network 28: Sentido inverso: nxt descarga activa
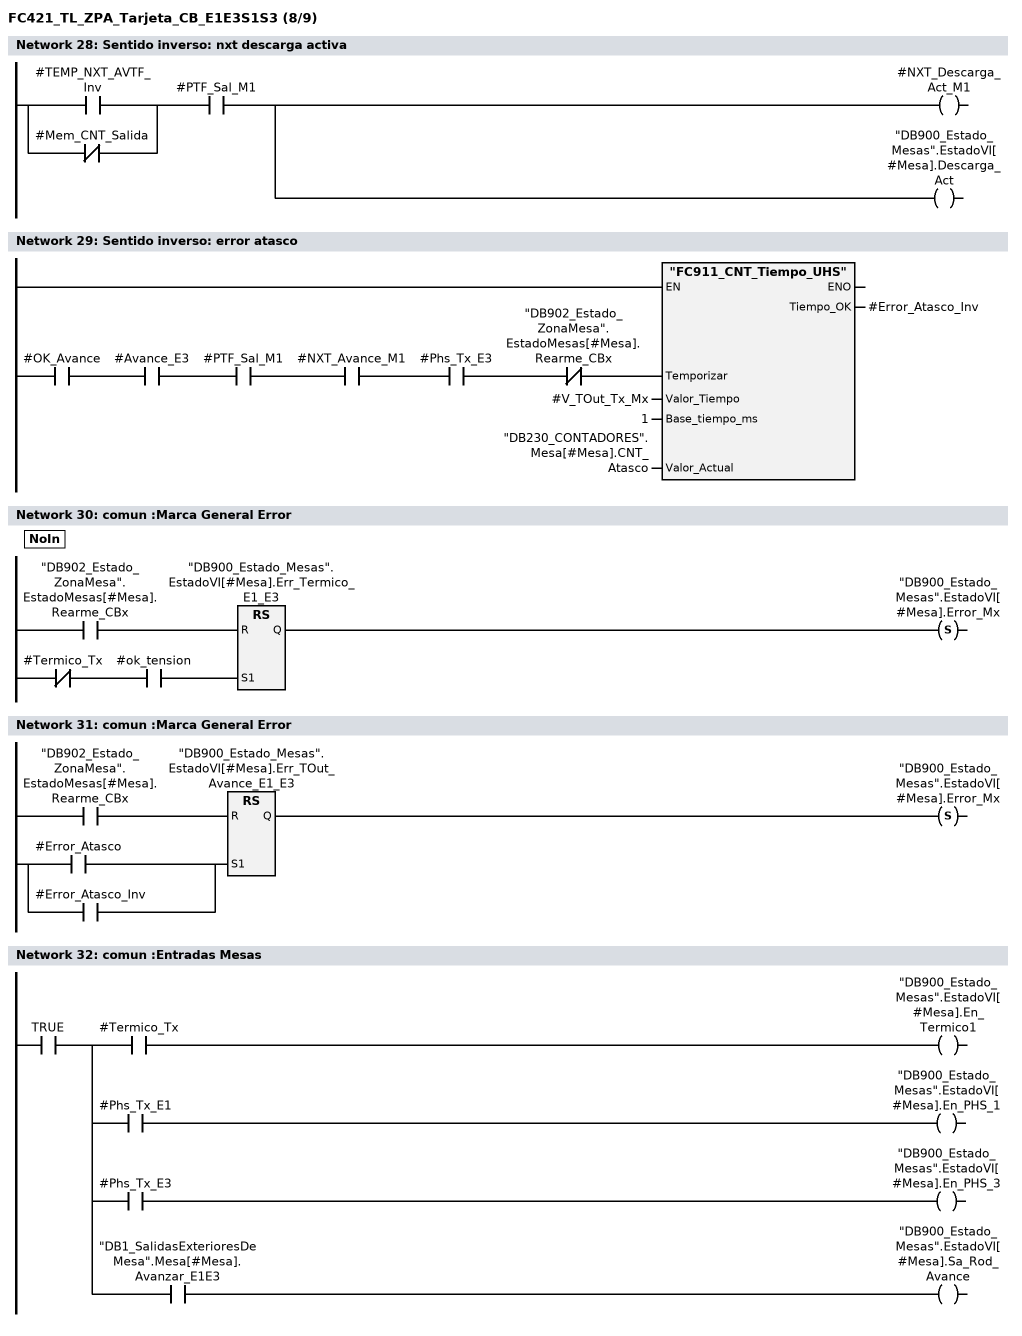
   RUNG wire#powerrail
      Contact( #TEMP_NXT_AVTF_Inv )
      wire#w1
      Contact( #PTF_Sal_M1 )
      wire#w2
      Coil( #NXT_Descarga_Act_M1 )
   END_RUNG
   RUNG wire#powerrail
      I_Contact( #Mem_CNT_Salida )
   END_RUNG wire#w1
   RUNG wire#w2
      Coil( "DB900_Estado_Mesas".EstadoVI[#Mesa].Descarga_Act )
   END_RUNG
   // the same network as SCL:
   #NXT_Descarga_Act_M1 := (#TEMP_NXT_AVTF_Inv OR NOT #Mem_CNT_Salida) AND #PTF_Sal_M1;
   "DB900_Estado_Mesas".EstadoVI[#Mesa].Descarga_Act := #NXT_Descarga_Act_M1;
END_REGION

REGION Network 29: Sentido inverso: error atasco
   RUNG wire#powerrail
      "FC911_CNT_Tiempo_UHS"(Temporizar := wire#w1, Valor_Tiempo := #V_TOut_Tx_Mx, Base_tiempo_ms := 1, Valor_Actual := "DB230_CONTADORES".Mesa[#Mesa].CNT_Atasco, Tiempo_OK => #Error_Atasco_Inv)
   END_RUNG
   RUNG wire#powerrail
      Contact( #OK_Avance )
      Contact( #Avance_E3 )
      Contact( #PTF_Sal_M1 )
      Contact( #NXT_Avance_M1 )
      Contact( #Phs_Tx_E3 )
      I_Contact( "DB902_Estado_ZonaMesa".EstadoMesas[#Mesa].Rearme_CBx )
   END_RUNG wire#w1
   // the same network as SCL:
   "FC911_CNT_Tiempo_UHS"(Temporizar := #OK_Avance AND #Avance_E3 AND #PTF_Sal_M1 AND #NXT_Avance_M1 AND #Phs_Tx_E3 AND NOT "DB902_Estado_ZonaMesa".EstadoMesas[#Mesa].Rearme_CBx,
                          Valor_Tiempo := #V_TOut_Tx_Mx,
                          Base_tiempo_ms := 1,
                          Valor_Actual := "DB230_CONTADORES".Mesa[#Mesa].CNT_Atasco,
                          Tiempo_OK => #Error_Atasco_Inv);
END_REGION

REGION Network 30: comun :Marca General Error
   Label( NoIn )
   RUNG wire#powerrail
      Contact( "DB902_Estado_ZonaMesa".EstadoMesas[#Mesa].Rearme_CBx )
      S_RS(operand := "DB900_Estado_Mesas".EstadoVI[#Mesa].Err_Termico_E1_E3, s1 := wire#w1)
      S_Coil( "DB900_Estado_Mesas".EstadoVI[#Mesa].Error_Mx )
   END_RUNG
   RUNG wire#powerrail
      I_Contact( #Termico_Tx )
      Contact( #ok_tension )
   END_RUNG wire#w1
   // the same network as SCL:
   NoIn:
   IF "DB902_Estado_ZonaMesa".EstadoMesas[#Mesa].Rearme_CBx THEN
       "DB900_Estado_Mesas".EstadoVI[#Mesa].Err_Termico_E1_E3 := FALSE;   // RS flip-flop
   END_IF;
   IF NOT #Termico_Tx AND #ok_tension THEN
       "DB900_Estado_Mesas".EstadoVI[#Mesa].Err_Termico_E1_E3 := TRUE;
   END_IF;
   IF "DB900_Estado_Mesas".EstadoVI[#Mesa].Err_Termico_E1_E3 THEN
       "DB900_Estado_Mesas".EstadoVI[#Mesa].Error_Mx := TRUE;
   END_IF;
END_REGION

REGION Network 31: comun :Marca General Error
   RUNG wire#powerrail
      Contact( "DB902_Estado_ZonaMesa".EstadoMesas[#Mesa].Rearme_CBx )
      S_RS(operand := "DB900_Estado_Mesas".EstadoVI[#Mesa].Err_TOut_Avance_E1_E3, s1 := wire#w1)
      S_Coil( "DB900_Estado_Mesas".EstadoVI[#Mesa].Error_Mx )
   END_RUNG
   RUNG wire#powerrail
      Contact( #Error_Atasco )
   END_RUNG wire#w1
   RUNG wire#powerrail
      Contact( #Error_Atasco_Inv )
   END_RUNG wire#w1
   // the same network as SCL:
   IF "DB902_Estado_ZonaMesa".EstadoMesas[#Mesa].Rearme_CBx THEN
       "DB900_Estado_Mesas".EstadoVI[#Mesa].Err_TOut_Avance_E1_E3 := FALSE;   // RS flip-flop
   END_IF;
   IF #Error_Atasco OR #Error_Atasco_Inv THEN
       "DB900_Estado_Mesas".EstadoVI[#Mesa].Err_TOut_Avance_E1_E3 := TRUE;
   END_IF;
   IF "DB900_Estado_Mesas".EstadoVI[#Mesa].Err_TOut_Avance_E1_E3 THEN
       "DB900_Estado_Mesas".EstadoVI[#Mesa].Error_Mx := TRUE;
   END_IF;
END_REGION

REGION Network 32: comun :Entradas Mesas
   RUNG wire#powerrail
      Contact( TRUE )
      wire#w1
      Contact( #Termico_Tx )
      Coil( "DB900_Estado_Mesas".EstadoVI[#Mesa].En_Termico1 )
   END_RUNG
   RUNG wire#w1
      Contact( #Phs_Tx_E1 )
      Coil( "DB900_Estado_Mesas".EstadoVI[#Mesa].En_PHS_1 )
   END_RUNG
   RUNG wire#w1
      Contact( #Phs_Tx_E3 )
      Coil( "DB900_Estado_Mesas".EstadoVI[#Mesa].En_PHS_3 )
   END_RUNG
   RUNG wire#w1
      Contact( "DB1_SalidasExterioresDeMesa".Mesa[#Mesa].Avanzar_E1E3 )
      Coil( "DB900_Estado_Mesas".EstadoVI[#Mesa].Sa_Rod_Avance )
   END_RUNG
   // the same network as SCL:
   "DB900_Estado_Mesas".EstadoVI[#Mesa].En_Termico1 := TRUE AND #Termico_Tx;
   "DB900_Estado_Mesas".EstadoVI[#Mesa].En_PHS_1 := TRUE AND #Phs_Tx_E1;
   "DB900_Estado_Mesas".EstadoVI[#Mesa].En_PHS_3 := TRUE AND #Phs_Tx_E3;
   "DB900_Estado_Mesas".EstadoVI[#Mesa].Sa_Rod_Avance := TRUE AND "DB1_SalidasExterioresDeMesa".Mesa[#Mesa].Avanzar_E1E3;
END_REGION

REGION Network 33: comun : ESTADOS MESA 1
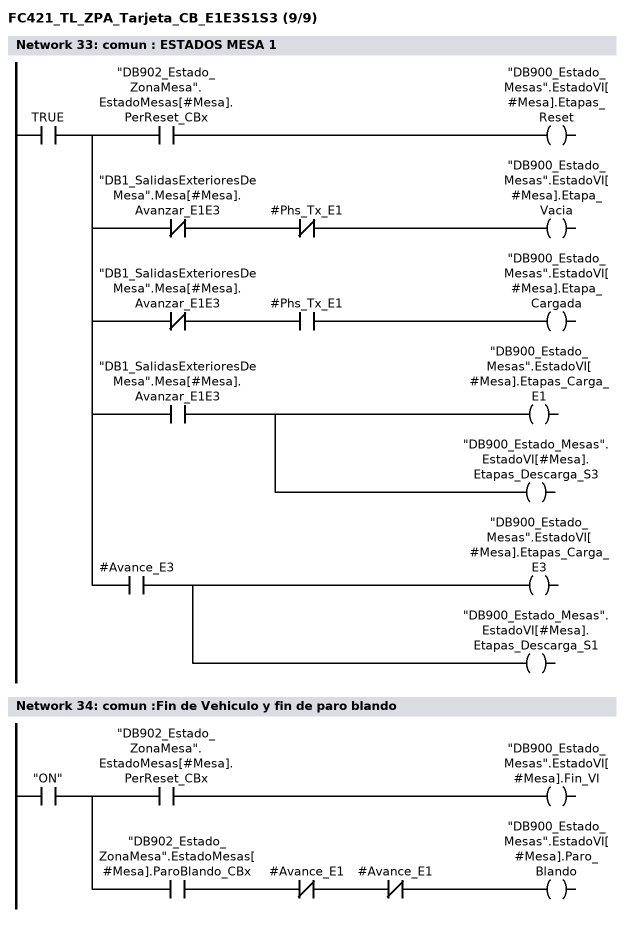
   RUNG wire#powerrail
      Contact( TRUE )
      wire#w1
      Contact( "DB902_Estado_ZonaMesa".EstadoMesas[#Mesa].PerReset_CBx )
      Coil( "DB900_Estado_Mesas".EstadoVI[#Mesa].Etapas_Reset )
   END_RUNG
   RUNG wire#w1
      I_Contact( "DB1_SalidasExterioresDeMesa".Mesa[#Mesa].Avanzar_E1E3 )
      I_Contact( #Phs_Tx_E1 )
      Coil( "DB900_Estado_Mesas".EstadoVI[#Mesa].Etapa_Vacia )
   END_RUNG
   RUNG wire#w1
      I_Contact( "DB1_SalidasExterioresDeMesa".Mesa[#Mesa].Avanzar_E1E3 )
      Contact( #Phs_Tx_E1 )
      Coil( "DB900_Estado_Mesas".EstadoVI[#Mesa].Etapa_Cargada )
   END_RUNG
   RUNG wire#w1
      Contact( "DB1_SalidasExterioresDeMesa".Mesa[#Mesa].Avanzar_E1E3 )
      wire#w2
      Coil( "DB900_Estado_Mesas".EstadoVI[#Mesa].Etapas_Carga_E1 )
   END_RUNG
   RUNG wire#w2
      Coil( "DB900_Estado_Mesas".EstadoVI[#Mesa].Etapas_Descarga_S3 )
   END_RUNG
   RUNG wire#w1
      Contact( #Avance_E3 )
      wire#w3
      Coil( "DB900_Estado_Mesas".EstadoVI[#Mesa].Etapas_Carga_E3 )
   END_RUNG
   RUNG wire#w3
      Coil( "DB900_Estado_Mesas".EstadoVI[#Mesa].Etapas_Descarga_S1 )
   END_RUNG
   // the same network as SCL:
   "DB900_Estado_Mesas".EstadoVI[#Mesa].Etapas_Reset := TRUE AND "DB902_Estado_ZonaMesa".EstadoMesas[#Mesa].PerReset_CBx;
   "DB900_Estado_Mesas".EstadoVI[#Mesa].Etapa_Vacia := TRUE AND NOT "DB1_SalidasExterioresDeMesa".Mesa[#Mesa].Avanzar_E1E3 AND NOT #Phs_Tx_E1;
   "DB900_Estado_Mesas".EstadoVI[#Mesa].Etapa_Cargada := TRUE AND NOT "DB1_SalidasExterioresDeMesa".Mesa[#Mesa].Avanzar_E1E3 AND #Phs_Tx_E1;
   #_w1 := TRUE AND "DB1_SalidasExterioresDeMesa".Mesa[#Mesa].Avanzar_E1E3;
   "DB900_Estado_Mesas".EstadoVI[#Mesa].Etapas_Carga_E1 := TRUE AND "DB1_SalidasExterioresDeMesa".Mesa[#Mesa].Avanzar_E1E3;
   "DB900_Estado_Mesas".EstadoVI[#Mesa].Etapas_Descarga_S3 := #_w1;
   "DB900_Estado_Mesas".EstadoVI[#Mesa].Etapas_Carga_E3 := TRUE AND #Avance_E3;
   "DB900_Estado_Mesas".EstadoVI[#Mesa].Etapas_Descarga_S1 := TRUE AND #Avance_E3;
END_REGION

REGION Network 34: comun :Fin de Vehiculo y fin de paro blando
   RUNG wire#powerrail
      Contact( "ON" )
      wire#w1
      Contact( "DB902_Estado_ZonaMesa".EstadoMesas[#Mesa].PerReset_CBx )
      Coil( "DB900_Estado_Mesas".EstadoVI[#Mesa].Fin_VI )
   END_RUNG
   RUNG wire#w1
      Contact( "DB902_Estado_ZonaMesa".EstadoMesas[#Mesa].ParoBlando_CBx )
      I_Contact( #Avance_E1 )
      I_Contact( #Avance_E1 )
      Coil( "DB900_Estado_Mesas".EstadoVI[#Mesa].Paro_Blando )
   END_RUNG
   // the same network as SCL:
   "DB900_Estado_Mesas".EstadoVI[#Mesa].Fin_VI := "ON" AND "DB902_Estado_ZonaMesa".EstadoMesas[#Mesa].PerReset_CBx;
   "DB900_Estado_Mesas".EstadoVI[#Mesa].Paro_Blando := "ON" AND "DB902_Estado_ZonaMesa".EstadoMesas[#Mesa].ParoBlando_CBx AND NOT #Avance_E1 AND NOT #Avance_E1;
END_REGION
END_FUNCTION
